(* IEC 61131-3 sources: RAG_PLC/data/result/test/060, 2 files *)

(* ---- wrapped.st ---- *)
(* =========================================================
   Generated by PLC-Eval Benchmark Wrapper
   ========================================================= *)

FUNCTION_BLOCK LLM_Wrapper_FB
VAR_INPUT
    I1 : BOOL;
    I2 : BOOL;
    TL : TIME;
END_VAR

VAR_OUTPUT
    Q1 : BOOL;
    Q2 : BOOL;
END_VAR

VAR
    T1 : TOF;
    T2 : TOF;
END_VAR

(*@KEY@: WORKSHEET
NAME: INTERLOCK
IEC_LANGUAGE: ST
*)
(* 输入信号有一个运行延迟，用于锁定另一个输入 *)
T1(IN := I1, PT := TL);
T2(IN := I2, PT := TL);

Q1 := I1 AND NOT T2.Q;
Q2 := I2 AND NOT T1.Q;
END_FUNCTION_BLOCK

PROGRAM Auto_Proxy_Prg
  VAR
    instance : LLM_Wrapper_FB;
  END_VAR

  instance();
END_PROGRAM

CONFIGURATION Config0
  RESOURCE Res0 ON PLC
    TASK TaskMain(INTERVAL := T#20ms, PRIORITY := 0);
    PROGRAM Inst0 WITH TaskMain : Auto_Proxy_Prg;
  END_RESOURCE
END_CONFIGURATION

(* ---- raw_code.st ---- *)
VAR_INPUT
    I1 : BOOL;
    I2 : BOOL;
    TL : TIME;
END_VAR

VAR_OUTPUT
    Q1 : BOOL;
    Q2 : BOOL;
END_VAR

VAR
    T1 : TOF;
    T2 : TOF;
END_VAR

(*@KEY@: WORKSHEET
NAME: INTERLOCK
IEC_LANGUAGE: ST
*)
(* 输入信号有一个运行延迟，用于锁定另一个输入 *)
T1(IN := I1, PT := TL);
T2(IN := I2, PT := TL);

Q1 := I1 AND NOT T2.Q;
Q2 := I2 AND NOT T1.Q;
